FUNCTION_BLOCK T2_Counter (* Basic Function Block Type *)
  (* Standard: 61499-2 *)
  (* Version 0.0, 2014-07-10, 4DIAC-IDE, 4DIAC-Consortium *)
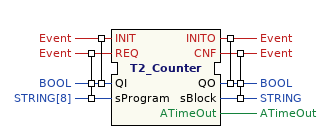
  EVENT_INPUT
    INIT WITH QI; (* Initialization Request *)
    REQ WITH QI, sProgram; (* Normal Execution Request *)
  END_EVENT
  EVENT_OUTPUT
    INITO WITH QO; (* Initialization Confirm *)
    CNF WITH QO, sBlock; (* Execution Confirmation *)
  END_EVENT
  VAR_INPUT
    QI : BOOL := TRUE; (* Input event qualifier *)
    sProgram : ARRAY [0..7] OF STRING := [0,0,0,0,0,0,0,0]; (* String array holding the blocks to be executed *)
  END_VAR
  VAR_OUTPUT
    QO : BOOL; (* Output event qualifier *)
    sBlock : STRING := Empty; (* String containing the next block to be executed *)
  END_VAR
  PLUGS
    ATimeOut : ATimeOut;
  END_PLUGS
  VAR
    Ins_Counter : INT := 0; (* Instruction counter *)
  END_VAR
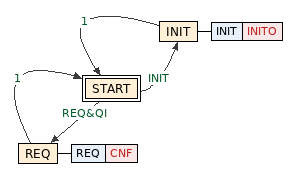
  EC_STATES
    START; (* Initial State *)
    INIT : INIT -> INITO; (* Initialization *)
    REQ : REQ -> CNF; (* Normal execution *)
  END_STATES
  EC_TRANSITIONS
    START TO INIT := INIT;
    INIT TO START := 1;
    START TO REQ := REQ&QI;
    REQ TO START := 1;
  END_TRANSITIONS
  ALGORITHM INIT IN ST: (* Initialization algorithm *)
QI := TRUE;
Ins_Counter := 0;
  END_ALGORITHM
  ALGORITHM REQ IN AnyText: (* Normally executed algorithm *)

  END_ALGORITHM
END_FUNCTION_BLOCK
